(* Logix 5000 project; controller PRU vendor 1 type 14 code 107 rev 20.13; software revision 20.01; part 8 of 17 *)
(* tags used below, declared in another part *)
   AFI : BOOL;
   Agilyx_KnifeGateIgnorePB : BOOL;
   COOL_MESSAGE_FON1 : TIMER;
   COOL_MESSAGE_FON2 : TIMER;
   COOL_VFD_Message : MESSAGE;
   DRYER : DUAL_SCREW;
   FAULT : DINT[100];
   FAULT_TIMER : TIMER[10000];
   FAULTS_FA4_IOK : BOOL;   // HI TEMP FAULTS ARE OK.
   FAULTS_FA4A_IOK : BOOL;   // HIGH TEMPERATURE FAULTS ARE OK.
   FAULTS_FA5A_IOK : BOOL;   // COOLING SCREW FAULTS ARE OK.
   FAULTS_FA5C_IOK : BOOL;   // KG021 FAULTS ARE OK.
   FAULTS_FA5D_IOK : BOOL;   // KG021 FAULTS ARE OK.
   HMI_ALARM_RESET : BOOL;
   K0621_ALARM_ION : BOOL;
   K0621_IS_CLOSED : BOOL;
   K0621_IS_OPEN : BOOL;
   K0622_ALARM_ION : BOOL;
   K0622_IS_CLOSED : BOOL;
   K0622_IS_OPEN : BOOL;
   K6021_GO_CLOSE_GON : BOOL;
   K6021_GO_OPEN_GON : BOOL;
   K6022_GO_CLOSE_GON : BOOL;
   K6022_GO_OPEN_GON : BOOL;
   Module_COOL_Fault : DINT;
   Module_COOL_Iok : BOOL;
   Module_COOL_Status : DINT;
   TE0101 : REAL;
   TE0102 : REAL;
   TE0103 : REAL;
   TE0104 : REAL;
   TE0105 : REAL;
   TE0106 : REAL;
   TE0107 : REAL;
   TE0108 : REAL;
   TE0109 : REAL;
   TE0110 : REAL;
   TE0111 : REAL;
   TE0112 : REAL;
   TE0113 : REAL;
   TE0114 : REAL;
   TE0115 : REAL;
   TE0116 : REAL;
   TE0117 : REAL;
   TE0118 : REAL;
   TE0119 : REAL;
   TE0120 : REAL;
   TE0121 : REAL;
   TE0122 : REAL;
   TE0123 : REAL;
   TE0124 : REAL;
   TE0125 : REAL;
   TE0126 : REAL;
   TE0127 : REAL;
   TE0128 : REAL;
   TE0129 : REAL;
   TE0130 : REAL;
   TE0201 : REAL;
   TE0202 : REAL;
   THRESHOLD : REAL[9000];
   VFD_3_Current_Real : REAL;
(* MainProgram, continued *)

ROUTINE B04_FAULTS_FA4_A_HIGH_TEMP_4000   (* ladder *)
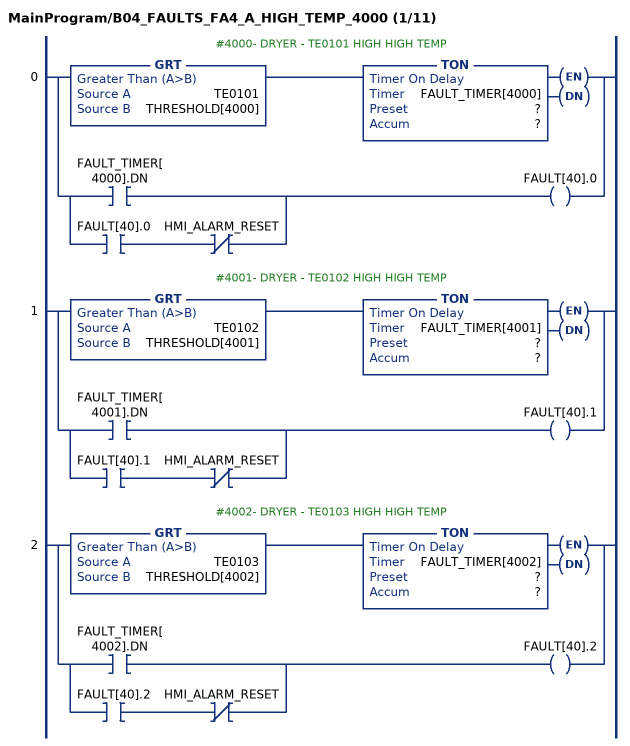
   // #4000- DRYER - TE0101 HIGH HIGH TEMP
   0: [GRT(TE0101,THRESHOLD[4000]) TON(FAULT_TIMER[4000],?,?) ,[XIC(FAULT_TIMER[4000].DN) ,XIC(FAULT[40].0) XIO(HMI_ALARM_RESET) ] OTE(FAULT[40].0) ];
   // #4001- DRYER - TE0102 HIGH HIGH TEMP
   1: [GRT(TE0102,THRESHOLD[4001]) TON(FAULT_TIMER[4001],?,?) ,[XIC(FAULT_TIMER[4001].DN) ,XIC(FAULT[40].1) XIO(HMI_ALARM_RESET) ] OTE(FAULT[40].1) ];
   // #4002- DRYER - TE0103 HIGH HIGH TEMP
   2: [GRT(TE0103,THRESHOLD[4002]) TON(FAULT_TIMER[4002],?,?) ,[XIC(FAULT_TIMER[4002].DN) ,XIC(FAULT[40].2) XIO(HMI_ALARM_RESET) ] OTE(FAULT[40].2) ];
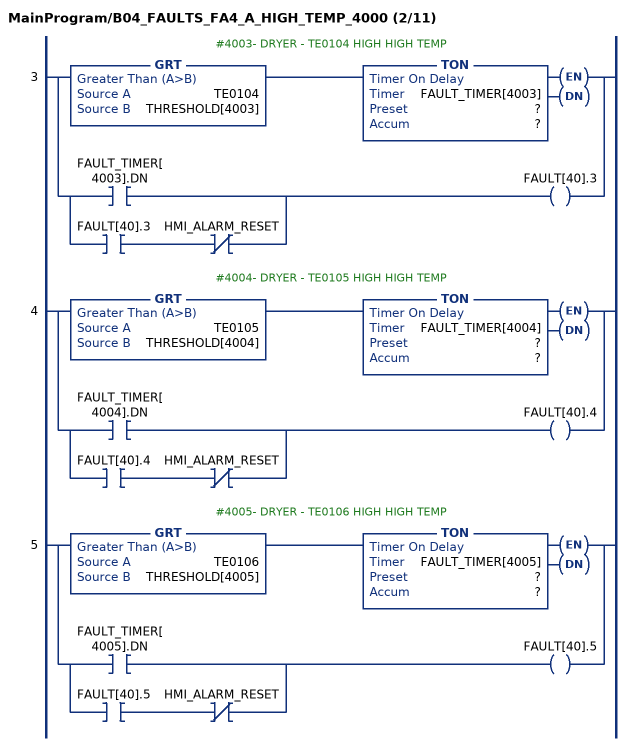
   // #4003- DRYER - TE0104 HIGH HIGH TEMP
   3: [GRT(TE0104,THRESHOLD[4003]) TON(FAULT_TIMER[4003],?,?) ,[XIC(FAULT_TIMER[4003].DN) ,XIC(FAULT[40].3) XIO(HMI_ALARM_RESET) ] OTE(FAULT[40].3) ];
   // #4004- DRYER - TE0105 HIGH HIGH TEMP
   4: [GRT(TE0105,THRESHOLD[4004]) TON(FAULT_TIMER[4004],?,?) ,[XIC(FAULT_TIMER[4004].DN) ,XIC(FAULT[40].4) XIO(HMI_ALARM_RESET) ] OTE(FAULT[40].4) ];
   // #4005- DRYER - TE0106 HIGH HIGH TEMP
   5: [GRT(TE0106,THRESHOLD[4005]) TON(FAULT_TIMER[4005],?,?) ,[XIC(FAULT_TIMER[4005].DN) ,XIC(FAULT[40].5) XIO(HMI_ALARM_RESET) ] OTE(FAULT[40].5) ];
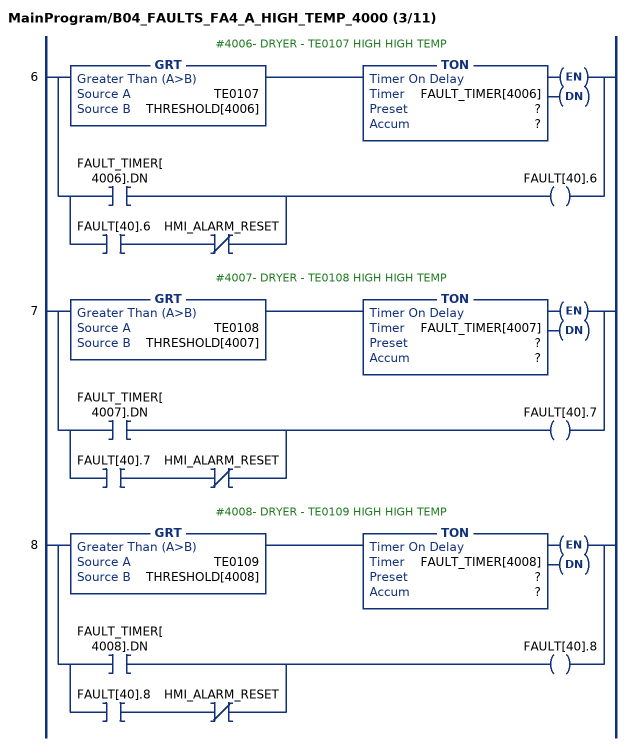
   // #4006- DRYER - TE0107 HIGH HIGH TEMP
   6: [GRT(TE0107,THRESHOLD[4006]) TON(FAULT_TIMER[4006],?,?) ,[XIC(FAULT_TIMER[4006].DN) ,XIC(FAULT[40].6) XIO(HMI_ALARM_RESET) ] OTE(FAULT[40].6) ];
   // #4007- DRYER - TE0108 HIGH HIGH TEMP
   7: [GRT(TE0108,THRESHOLD[4007]) TON(FAULT_TIMER[4007],?,?) ,[XIC(FAULT_TIMER[4007].DN) ,XIC(FAULT[40].7) XIO(HMI_ALARM_RESET) ] OTE(FAULT[40].7) ];
   // #4008- DRYER - TE0109 HIGH HIGH TEMP
   8: [GRT(TE0109,THRESHOLD[4008]) TON(FAULT_TIMER[4008],?,?) ,[XIC(FAULT_TIMER[4008].DN) ,XIC(FAULT[40].8) XIO(HMI_ALARM_RESET) ] OTE(FAULT[40].8) ];
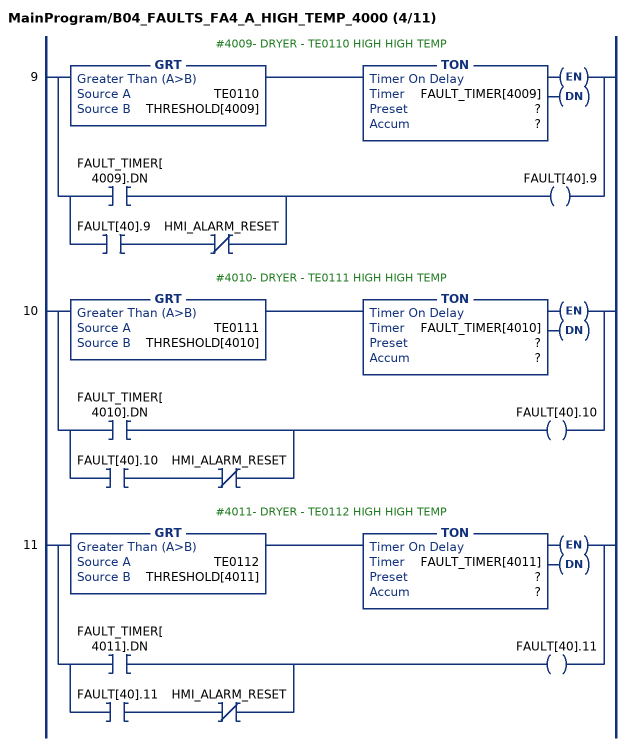
   // #4009- DRYER - TE0110 HIGH HIGH TEMP
   9: [GRT(TE0110,THRESHOLD[4009]) TON(FAULT_TIMER[4009],?,?) ,[XIC(FAULT_TIMER[4009].DN) ,XIC(FAULT[40].9) XIO(HMI_ALARM_RESET) ] OTE(FAULT[40].9) ];
   // #4010- DRYER - TE0111 HIGH HIGH TEMP
   10: [GRT(TE0111,THRESHOLD[4010]) TON(FAULT_TIMER[4010],?,?) ,[XIC(FAULT_TIMER[4010].DN) ,XIC(FAULT[40].10) XIO(HMI_ALARM_RESET) ] OTE(FAULT[40].10) ];
   // #4011- DRYER - TE0112 HIGH HIGH TEMP
   11: [GRT(TE0112,THRESHOLD[4011]) TON(FAULT_TIMER[4011],?,?) ,[XIC(FAULT_TIMER[4011].DN) ,XIC(FAULT[40].11) XIO(HMI_ALARM_RESET) ] OTE(FAULT[40].11) ];
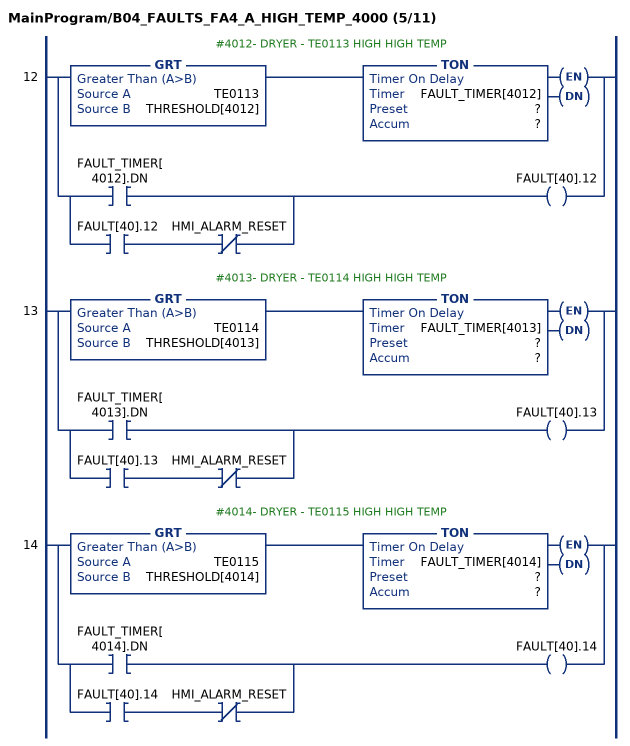
   // #4012- DRYER - TE0113 HIGH HIGH TEMP
   12: [GRT(TE0113,THRESHOLD[4012]) TON(FAULT_TIMER[4012],?,?) ,[XIC(FAULT_TIMER[4012].DN) ,XIC(FAULT[40].12) XIO(HMI_ALARM_RESET) ] OTE(FAULT[40].12) ];
   // #4013- DRYER - TE0114 HIGH HIGH TEMP
   13: [GRT(TE0114,THRESHOLD[4013]) TON(FAULT_TIMER[4013],?,?) ,[XIC(FAULT_TIMER[4013].DN) ,XIC(FAULT[40].13) XIO(HMI_ALARM_RESET) ] OTE(FAULT[40].13) ];
   // #4014- DRYER - TE0115 HIGH HIGH TEMP
   14: [GRT(TE0115,THRESHOLD[4014]) TON(FAULT_TIMER[4014],?,?) ,[XIC(FAULT_TIMER[4014].DN) ,XIC(FAULT[40].14) XIO(HMI_ALARM_RESET) ] OTE(FAULT[40].14) ];
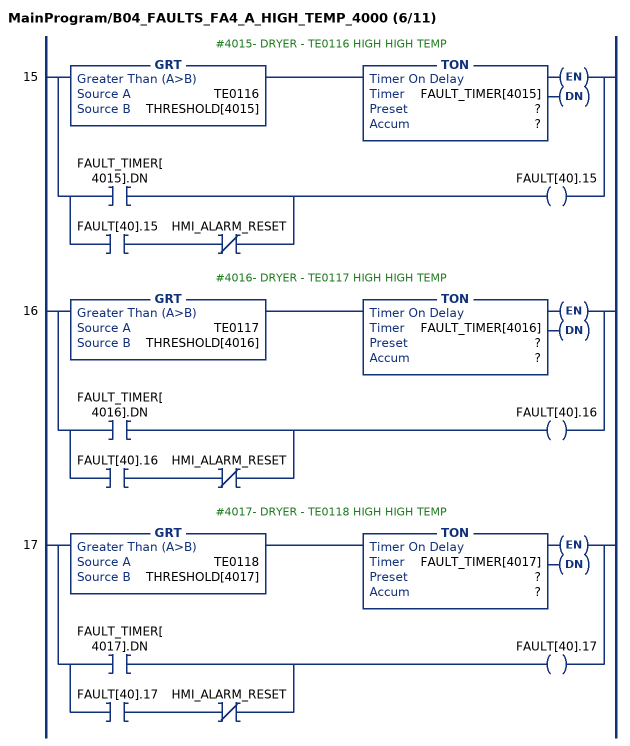
   // #4015- DRYER - TE0116 HIGH HIGH TEMP
   15: [GRT(TE0116,THRESHOLD[4015]) TON(FAULT_TIMER[4015],?,?) ,[XIC(FAULT_TIMER[4015].DN) ,XIC(FAULT[40].15) XIO(HMI_ALARM_RESET) ] OTE(FAULT[40].15) ];
   // #4016- DRYER - TE0117 HIGH HIGH TEMP
   16: [GRT(TE0117,THRESHOLD[4016]) TON(FAULT_TIMER[4016],?,?) ,[XIC(FAULT_TIMER[4016].DN) ,XIC(FAULT[40].16) XIO(HMI_ALARM_RESET) ] OTE(FAULT[40].16) ];
   // #4017- DRYER - TE0118 HIGH HIGH TEMP
   17: [GRT(TE0118,THRESHOLD[4017]) TON(FAULT_TIMER[4017],?,?) ,[XIC(FAULT_TIMER[4017].DN) ,XIC(FAULT[40].17) XIO(HMI_ALARM_RESET) ] OTE(FAULT[40].17) ];
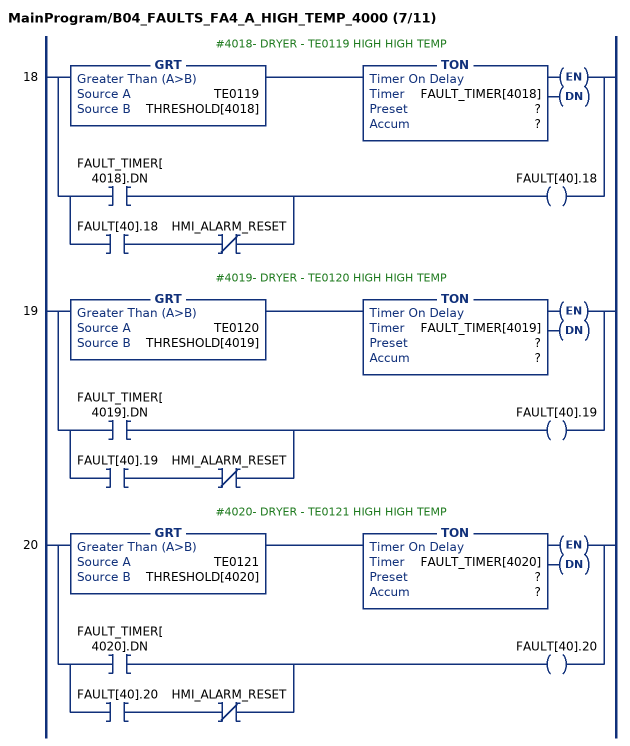
   // #4018- DRYER - TE0119 HIGH HIGH TEMP
   18: [GRT(TE0119,THRESHOLD[4018]) TON(FAULT_TIMER[4018],?,?) ,[XIC(FAULT_TIMER[4018].DN) ,XIC(FAULT[40].18) XIO(HMI_ALARM_RESET) ] OTE(FAULT[40].18) ];
   // #4019- DRYER - TE0120 HIGH HIGH TEMP
   19: [GRT(TE0120,THRESHOLD[4019]) TON(FAULT_TIMER[4019],?,?) ,[XIC(FAULT_TIMER[4019].DN) ,XIC(FAULT[40].19) XIO(HMI_ALARM_RESET) ] OTE(FAULT[40].19) ];
   // #4020- DRYER - TE0121 HIGH HIGH TEMP
   20: [GRT(TE0121,THRESHOLD[4020]) TON(FAULT_TIMER[4020],?,?) ,[XIC(FAULT_TIMER[4020].DN) ,XIC(FAULT[40].20) XIO(HMI_ALARM_RESET) ] OTE(FAULT[40].20) ];
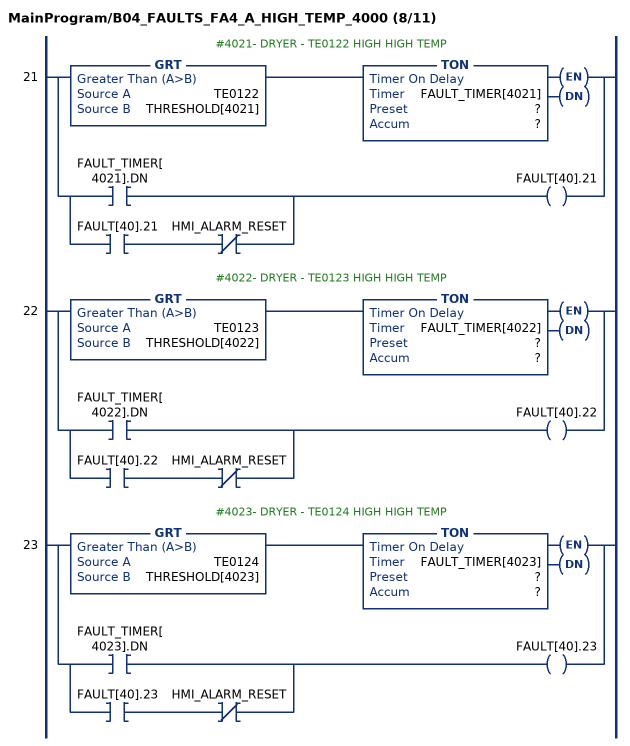
   // #4021- DRYER - TE0122 HIGH HIGH TEMP
   21: [GRT(TE0122,THRESHOLD[4021]) TON(FAULT_TIMER[4021],?,?) ,[XIC(FAULT_TIMER[4021].DN) ,XIC(FAULT[40].21) XIO(HMI_ALARM_RESET) ] OTE(FAULT[40].21) ];
   // #4022- DRYER - TE0123 HIGH HIGH TEMP
   22: [GRT(TE0123,THRESHOLD[4022]) TON(FAULT_TIMER[4022],?,?) ,[XIC(FAULT_TIMER[4022].DN) ,XIC(FAULT[40].22) XIO(HMI_ALARM_RESET) ] OTE(FAULT[40].22) ];
   // #4023- DRYER - TE0124 HIGH HIGH TEMP
   23: [GRT(TE0124,THRESHOLD[4023]) TON(FAULT_TIMER[4023],?,?) ,[XIC(FAULT_TIMER[4023].DN) ,XIC(FAULT[40].23) XIO(HMI_ALARM_RESET) ] OTE(FAULT[40].23) ];
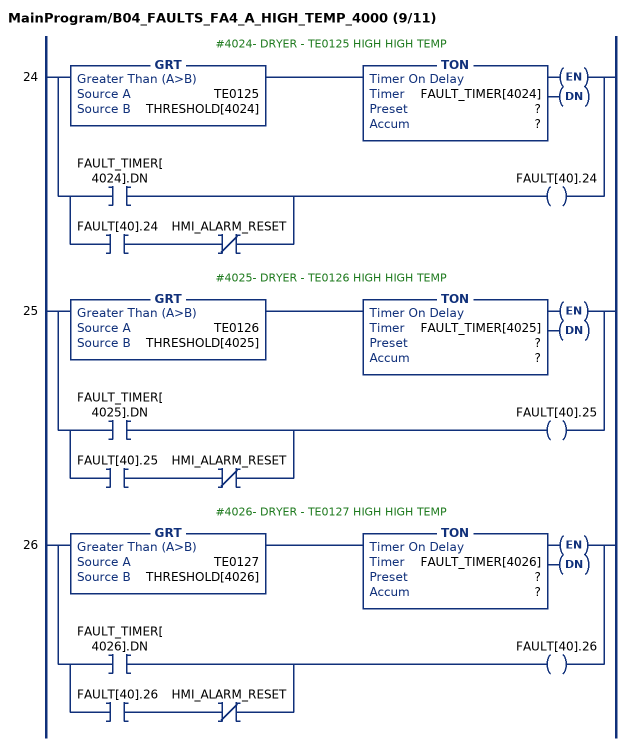
   // #4024- DRYER - TE0125 HIGH HIGH TEMP
   24: [GRT(TE0125,THRESHOLD[4024]) TON(FAULT_TIMER[4024],?,?) ,[XIC(FAULT_TIMER[4024].DN) ,XIC(FAULT[40].24) XIO(HMI_ALARM_RESET) ] OTE(FAULT[40].24) ];
   // #4025- DRYER - TE0126 HIGH HIGH TEMP
   25: [GRT(TE0126,THRESHOLD[4025]) TON(FAULT_TIMER[4025],?,?) ,[XIC(FAULT_TIMER[4025].DN) ,XIC(FAULT[40].25) XIO(HMI_ALARM_RESET) ] OTE(FAULT[40].25) ];
   // #4026- DRYER - TE0127 HIGH HIGH TEMP
   26: [GRT(TE0127,THRESHOLD[4026]) TON(FAULT_TIMER[4026],?,?) ,[XIC(FAULT_TIMER[4026].DN) ,XIC(FAULT[40].26) XIO(HMI_ALARM_RESET) ] OTE(FAULT[40].26) ];
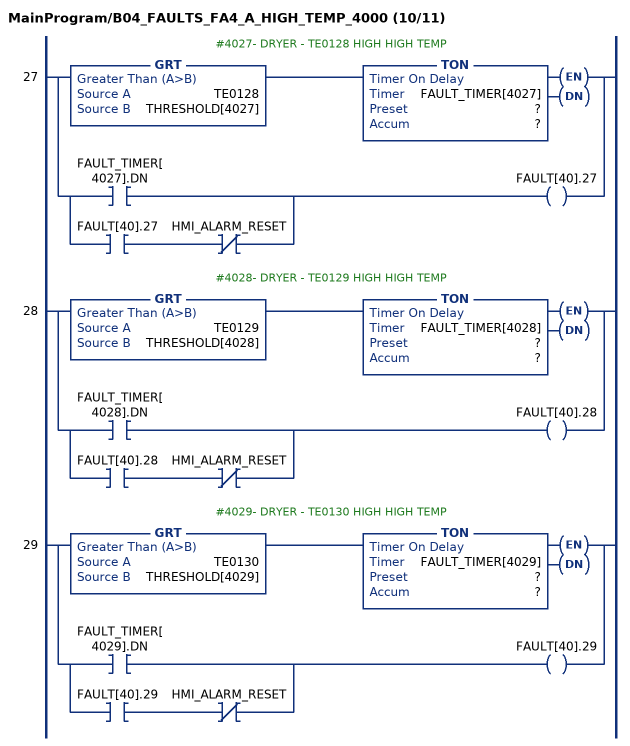
   // #4027- DRYER - TE0128 HIGH HIGH TEMP
   27: [GRT(TE0128,THRESHOLD[4027]) TON(FAULT_TIMER[4027],?,?) ,[XIC(FAULT_TIMER[4027].DN) ,XIC(FAULT[40].27) XIO(HMI_ALARM_RESET) ] OTE(FAULT[40].27) ];
   // #4028- DRYER - TE0129 HIGH HIGH TEMP
   28: [GRT(TE0129,THRESHOLD[4028]) TON(FAULT_TIMER[4028],?,?) ,[XIC(FAULT_TIMER[4028].DN) ,XIC(FAULT[40].28) XIO(HMI_ALARM_RESET) ] OTE(FAULT[40].28) ];
   // #4029- DRYER - TE0130 HIGH HIGH TEMP
   29: [GRT(TE0130,THRESHOLD[4029]) TON(FAULT_TIMER[4029],?,?) ,[XIC(FAULT_TIMER[4029].DN) ,XIC(FAULT[40].29) XIO(HMI_ALARM_RESET) ] OTE(FAULT[40].29) ];
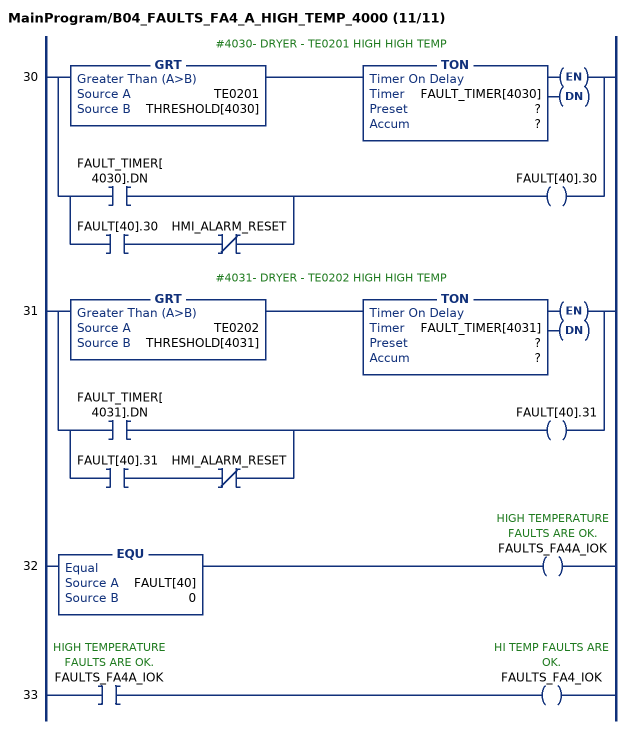
   // #4030- DRYER - TE0201 HIGH HIGH TEMP
   30: [GRT(TE0201,THRESHOLD[4030]) TON(FAULT_TIMER[4030],?,?) ,[XIC(FAULT_TIMER[4030].DN) ,XIC(FAULT[40].30) XIO(HMI_ALARM_RESET) ] OTE(FAULT[40].30) ];
   // #4031- DRYER - TE0202 HIGH HIGH TEMP
   31: [GRT(TE0202,THRESHOLD[4031]) TON(FAULT_TIMER[4031],?,?) ,[XIC(FAULT_TIMER[4031].DN) ,XIC(FAULT[40].31) XIO(HMI_ALARM_RESET) ] OTE(FAULT[40].31) ];
   32: EQU(FAULT[40],0)OTE(FAULTS_FA4A_IOK);
   33: XIC(FAULTS_FA4A_IOK)OTE(FAULTS_FA4_IOK);
END_ROUTINE

ROUTINE B05_FAULTS_FA5_A_COOLSCREW_5000   (* ladder *)
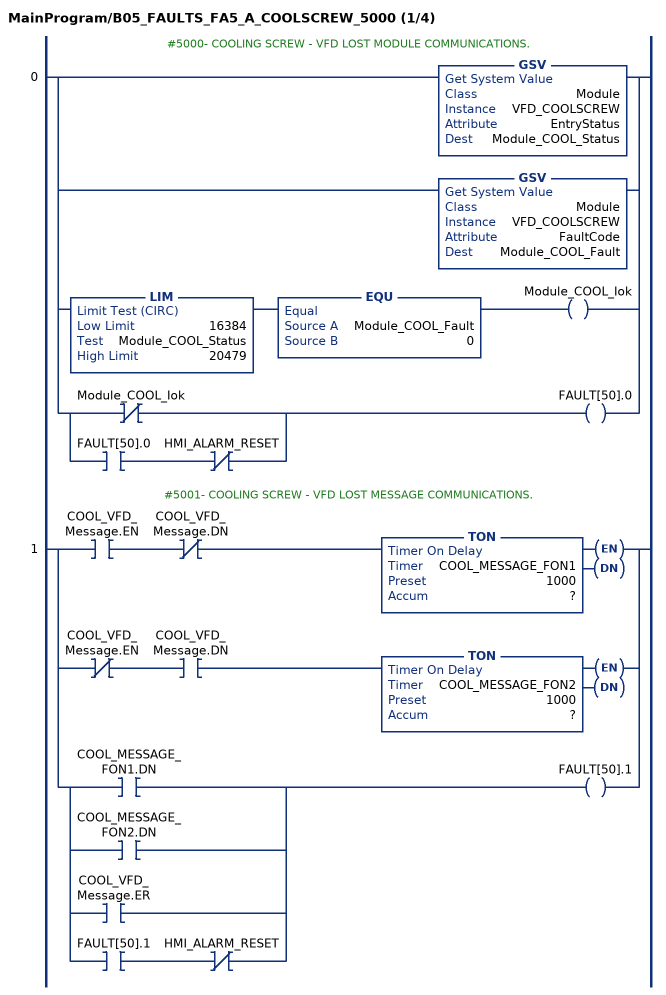
   // #5000- COOLING SCREW - VFD LOST MODULE COMMUNICATIONS.
   0: [GSV(Module,VFD_COOLSCREW,EntryStatus,Module_COOL_Status) ,GSV(Module,VFD_COOLSCREW,FaultCode,Module_COOL_Fault) ,LIM(16384,Module_COOL_Status,20479) EQU(Module_COOL_Fault,0) OTE(Module_COOL_Iok) ,[XIO(Module_COOL_Iok) ,XIC(FAULT[50].0) XIO(HMI_ALARM_RESET) ] OTE(FAULT[50].0) ];
   // #5001- COOLING SCREW - VFD LOST MESSAGE COMMUNICATIONS.
   1: [[XIC(COOL_VFD_Message.EN) XIO(COOL_VFD_Message.DN) TON(COOL_MESSAGE_FON1,?,?) ,XIO(COOL_VFD_Message.EN) XIC(COOL_VFD_Message.DN) TON(COOL_MESSAGE_FON2,?,?) ] ,[XIC(COOL_MESSAGE_FON1.DN) ,XIC(COOL_MESSAGE_FON2.DN) ,XIC(COOL_VFD_Message.ER) ,XIC(FAULT[50].1) XIO(HMI_ALARM_RESET) ] OTE(FAULT[50].1) ];
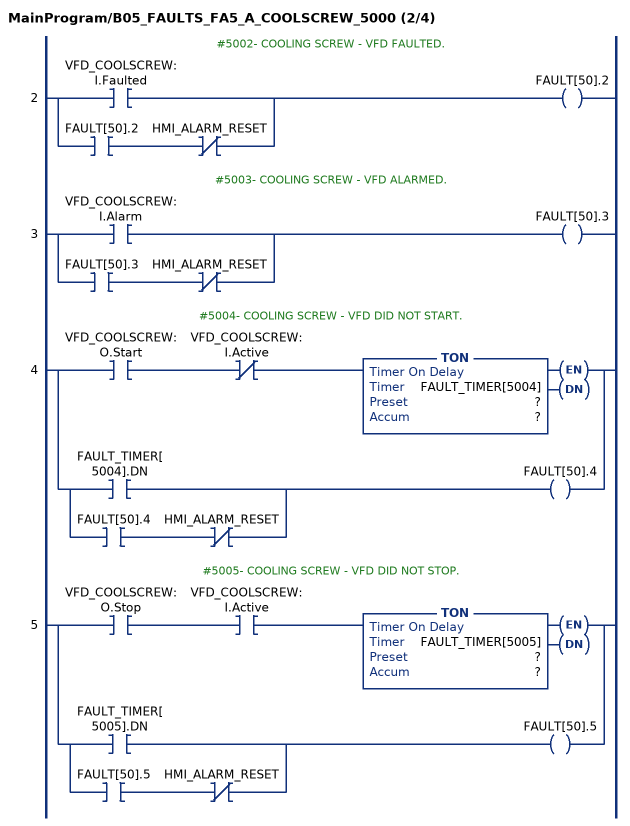
   // #5002- COOLING SCREW - VFD FAULTED.
   2: [XIC(VFD_COOLSCREW:I.Faulted) ,XIC(FAULT[50].2) XIO(HMI_ALARM_RESET) ]OTE(FAULT[50].2);
   // #5003- COOLING SCREW - VFD ALARMED.
   3: [XIC(VFD_COOLSCREW:I.Alarm) ,XIC(FAULT[50].3) XIO(HMI_ALARM_RESET) ]OTE(FAULT[50].3);
   // #5004- COOLING SCREW - VFD DID NOT START.
   4: [XIC(VFD_COOLSCREW:O.Start) XIO(VFD_COOLSCREW:I.Active) TON(FAULT_TIMER[5004],?,?) ,[XIC(FAULT_TIMER[5004].DN) ,XIC(FAULT[50].4) XIO(HMI_ALARM_RESET) ] OTE(FAULT[50].4) ];
   // #5005- COOLING SCREW - VFD DID NOT STOP.
   5: [XIC(VFD_COOLSCREW:O.Stop) XIC(VFD_COOLSCREW:I.Active) TON(FAULT_TIMER[5005],?,?) ,[XIC(FAULT_TIMER[5005].DN) ,XIC(FAULT[50].5) XIO(HMI_ALARM_RESET) ] OTE(FAULT[50].5) ];
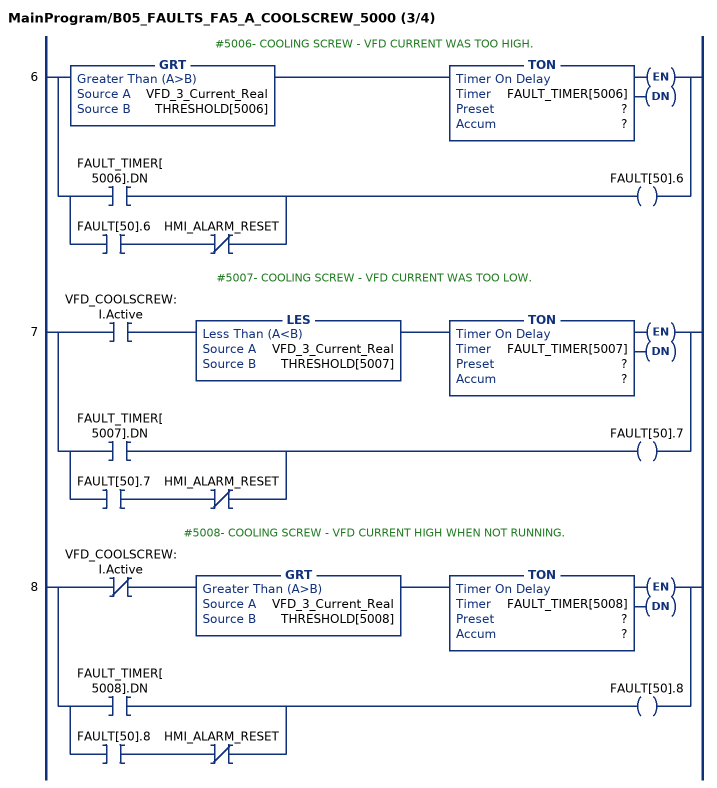
   // #5006- COOLING SCREW - VFD CURRENT WAS TOO HIGH.
   6: [GRT(VFD_3_Current_Real,THRESHOLD[5006]) TON(FAULT_TIMER[5006],?,?) ,[XIC(FAULT_TIMER[5006].DN) ,XIC(FAULT[50].6) XIO(HMI_ALARM_RESET) ] OTE(FAULT[50].6) ];
   // #5007- COOLING SCREW - VFD CURRENT WAS TOO LOW.
   7: [XIC(VFD_COOLSCREW:I.Active) LES(VFD_3_Current_Real,THRESHOLD[5007]) TON(FAULT_TIMER[5007],?,?) ,[XIC(FAULT_TIMER[5007].DN) ,XIC(FAULT[50].7) XIO(HMI_ALARM_RESET) ] OTE(FAULT[50].7) ];
   // #5008- COOLING SCREW - VFD CURRENT HIGH WHEN NOT RUNNING.
   8: [XIO(VFD_COOLSCREW:I.Active) GRT(VFD_3_Current_Real,THRESHOLD[5008]) TON(FAULT_TIMER[5008],?,?) ,[XIC(FAULT_TIMER[5008].DN) ,XIC(FAULT[50].8) XIO(HMI_ALARM_RESET) ] OTE(FAULT[50].8) ];
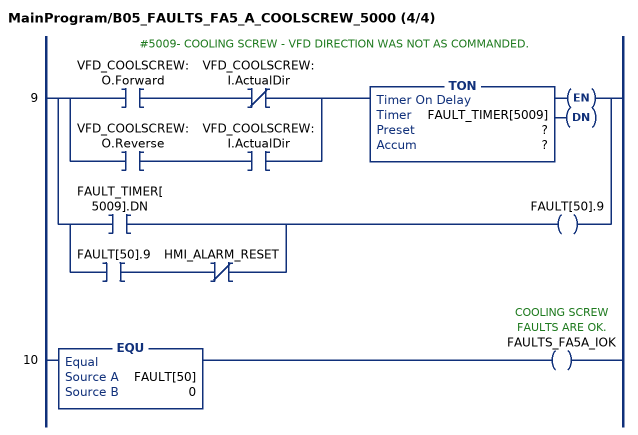
   // #5009- COOLING SCREW - VFD DIRECTION WAS NOT AS COMMANDED.
   9: [[XIC(VFD_COOLSCREW:O.Forward) XIO(VFD_COOLSCREW:I.ActualDir) ,XIC(VFD_COOLSCREW:O.Reverse) XIC(VFD_COOLSCREW:I.ActualDir) ] TON(FAULT_TIMER[5009],?,?) ,[XIC(FAULT_TIMER[5009].DN) ,XIC(FAULT[50].9) XIO(HMI_ALARM_RESET) ] OTE(FAULT[50].9) ];
   10: EQU(FAULT[50],0)OTE(FAULTS_FA5A_IOK);
END_ROUTINE

ROUTINE B05_FAULTS_FA5_C_KG021_6500   (* ladder *)
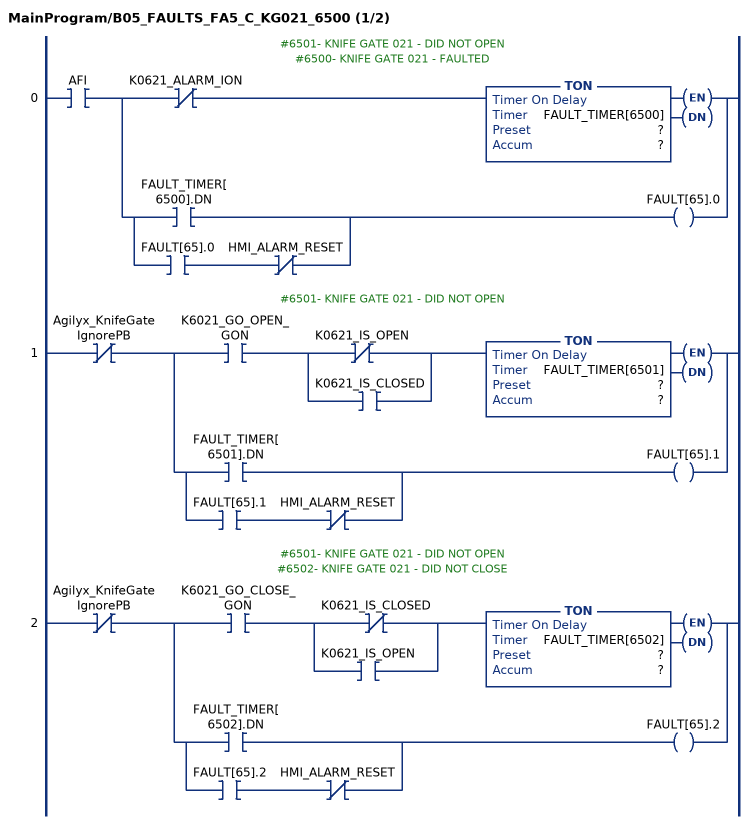
   // #6501- KNIFE GATE 021 - DID NOT OPEN
   // #6500- KNIFE GATE 021 - FAULTED
   0: XIC(AFI)[XIO(K0621_ALARM_ION) TON(FAULT_TIMER[6500],?,?) ,[XIC(FAULT_TIMER[6500].DN) ,XIC(FAULT[65].0) XIO(HMI_ALARM_RESET) ] OTE(FAULT[65].0) ];
   // #6501- KNIFE GATE 021 - DID NOT OPEN
   1: XIO(Agilyx_KnifeGateIgnorePB)[XIC(K6021_GO_OPEN_GON) [XIO(K0621_IS_OPEN) ,XIC(K0621_IS_CLOSED) ] TON(FAULT_TIMER[6501],?,?) ,[XIC(FAULT_TIMER[6501].DN) ,XIC(FAULT[65].1) XIO(HMI_ALARM_RESET) ] OTE(FAULT[65].1) ];
   // #6501- KNIFE GATE 021 - DID NOT OPEN
   // #6502- KNIFE GATE 021 - DID NOT CLOSE
   2: XIO(Agilyx_KnifeGateIgnorePB)[XIC(K6021_GO_CLOSE_GON) [XIO(K0621_IS_CLOSED) ,XIC(K0621_IS_OPEN) ] TON(FAULT_TIMER[6502],?,?) ,[XIC(FAULT_TIMER[6502].DN) ,XIC(FAULT[65].2) XIO(HMI_ALARM_RESET) ] OTE(FAULT[65].2) ];
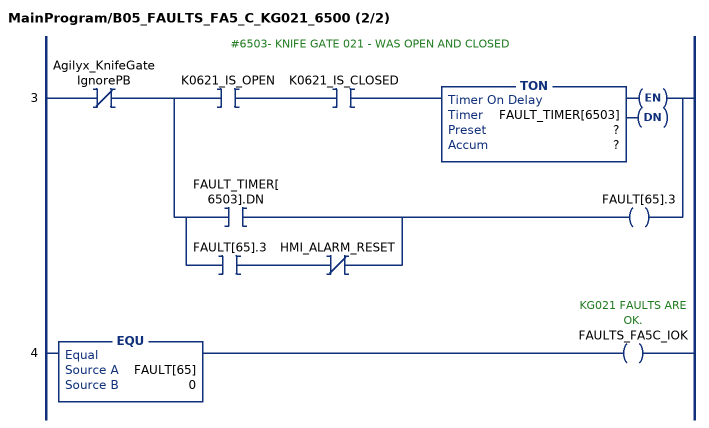
   // #6503- KNIFE GATE 021 - WAS OPEN AND CLOSED
   3: XIO(Agilyx_KnifeGateIgnorePB)[XIC(K0621_IS_OPEN) XIC(K0621_IS_CLOSED) TON(FAULT_TIMER[6503],?,?) ,[XIC(FAULT_TIMER[6503].DN) ,XIC(FAULT[65].3) XIO(HMI_ALARM_RESET) ] OTE(FAULT[65].3) ];
   4: EQU(FAULT[65],0)OTE(FAULTS_FA5C_IOK);
END_ROUTINE

ROUTINE B05_FAULTS_FA5_D_KG022_6600   (* ladder *)
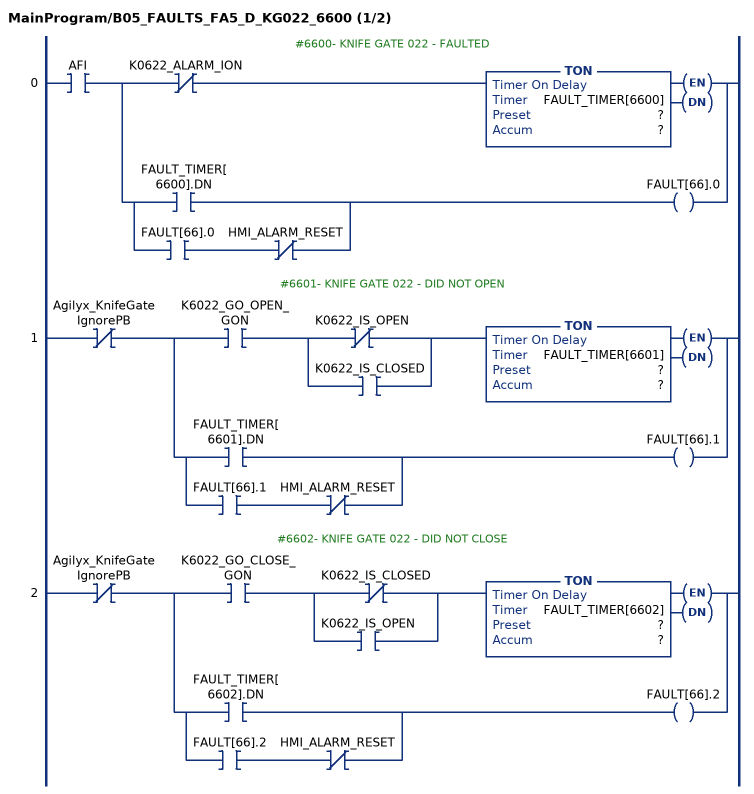
   // #6600- KNIFE GATE 022 - FAULTED
   0: XIC(AFI)[XIO(K0622_ALARM_ION) TON(FAULT_TIMER[6600],?,?) ,[XIC(FAULT_TIMER[6600].DN) ,XIC(FAULT[66].0) XIO(HMI_ALARM_RESET) ] OTE(FAULT[66].0) ];
   // #6601- KNIFE GATE 022 - DID NOT OPEN
   1: XIO(Agilyx_KnifeGateIgnorePB)[XIC(K6022_GO_OPEN_GON) [XIO(K0622_IS_OPEN) ,XIC(K0622_IS_CLOSED) ] TON(FAULT_TIMER[6601],?,?) ,[XIC(FAULT_TIMER[6601].DN) ,XIC(FAULT[66].1) XIO(HMI_ALARM_RESET) ] OTE(FAULT[66].1) ];
   // #6602- KNIFE GATE 022 - DID NOT CLOSE
   2: XIO(Agilyx_KnifeGateIgnorePB)[XIC(K6022_GO_CLOSE_GON) [XIO(K0622_IS_CLOSED) ,XIC(K0622_IS_OPEN) ] TON(FAULT_TIMER[6602],?,?) ,[XIC(FAULT_TIMER[6602].DN) ,XIC(FAULT[66].2) XIO(HMI_ALARM_RESET) ] OTE(FAULT[66].2) ];
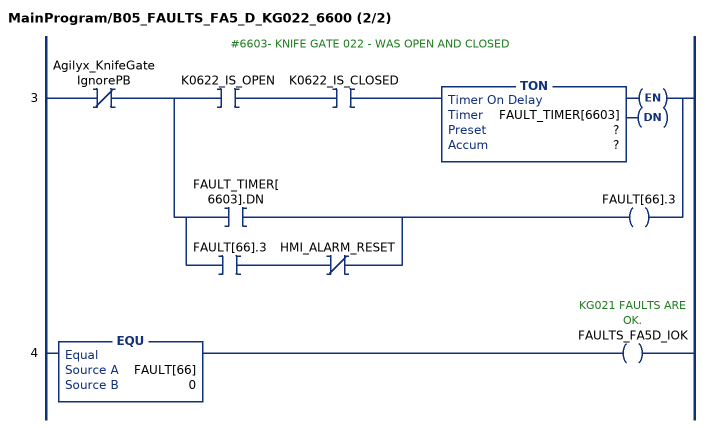
   // #6603- KNIFE GATE 022 - WAS OPEN AND CLOSED
   3: XIO(Agilyx_KnifeGateIgnorePB)[XIC(K0622_IS_OPEN) XIC(K0622_IS_CLOSED) TON(FAULT_TIMER[6603],?,?) ,[XIC(FAULT_TIMER[6603].DN) ,XIC(FAULT[66].3) XIO(HMI_ALARM_RESET) ] OTE(FAULT[66].3) ];
   4: EQU(FAULT[66],0)OTE(FAULTS_FA5D_IOK);
END_ROUTINE
